(* IEC 61131-3 sources: HappyLearnCodesys/content/softmotion/CustomKinematics_Implementation, 3 files *)

(* ---- Jog.st ---- *)
(*
    檔案用途：
      封裝一個 Jog 功能塊，讓使用者可以同時在「軸空間（ACS）」與「笛卡兒空間（MCS）」下
      以按鍵方式點動 Gantry3C 自訂運動學的 TCP 位置。
    教學重點：
      - 利用兩個 SMC_GroupJog2 實例（jog_mcs、jog_axes）分別處理 TCP Jog 與關節 Jog。
      - 理解來自視覺介面的按鍵輸入（Jog_TCP_*、Jog_Drive_*）如何對應到 Forward/Backward 陣列。
      - 作為「自訂運動學上層 Jog 介面」的範例，可套用到其他 kinematics。
*)
/// This FB combines jogging in both axis space as well as cartesian space.
/// It uses two instances of SMC_GroupJog2. One for axis space and the other for cartesian space.
/// This FB can be used along with the visu templates V_RobotPosition_axes
/// and V_RobotPosition_cart_Jog to jog any kinematics in cartesian and axis space.

FUNCTION_BLOCK Jog
VAR_IN_OUT
	/// Reference to Axisgroup
	AxisGroup : AXIS_GROUP_REF_SM3;
END_VAR
VAR_INPUT
	/// Inputs (from the visu) to jog the robot in cartesian space
	Jog_TCP_Xp : BOOL;
	Jog_TCP_Xn : BOOL;
	Jog_TCP_Yp : BOOL;
	Jog_TCP_Yn : BOOL;
	Jog_TCP_Zp : BOOL;
	Jog_TCP_Zn : BOOL;
	Jog_TCP_Ap : BOOL;
	Jog_TCP_An : BOOL;
	Jog_TCP_Bp : BOOL;
	Jog_TCP_Bn : BOOL;
	Jog_TCP_Cp : BOOL;
	Jog_TCP_Cn : BOOL;

	/// Inputs (from the visu) to jog the robot in axis space
	Jog_Drive_Xp : BOOL;
	Jog_Drive_Xn : BOOL;
	Jog_Drive_Yp : BOOL;
	Jog_Drive_Yn : BOOL;
	Jog_Drive_Zp : BOOL;
	Jog_Drive_Zn : BOOL;
	Jog_Drive_Cp : BOOL;
	Jog_Drive_Cn : BOOL;

END_VAR
VAR
	/// SMC_GroupJog2 for cartesian space
	jog_mcs : SMC_GroupJog2 :=(Enable := TRUE, MaxLinearDistance := 2, MaxAngularDistance := 1,
							VelFactor := 1, AccFactor := 1, JerkFactor := 1,
							Velocity := 100, Acceleration := 1000, Deceleration := 1000, Jerk := 1000,
						    CoordSystem:= SMC_COORD_SYSTEM.MCS);

	/// SMC_GroupJog2 for axes space
	jog_axes : SMC_GroupJog2 :=(Enable := TRUE, MaxLinearDistance := 2, MaxAngularDistance := 1,
							VelFactor := 1, AccFactor := 1, JerkFactor := 1,
							Velocity := 100, Acceleration := 1000, Deceleration := 1000, Jerk := 1000,
						    CoordSystem:= SMC_COORD_SYSTEM.ACS);
END_VAR

jog_mcs.Forward[0] := Jog_TCP_Xp;
jog_mcs.Forward[1] := Jog_TCP_Yp;
jog_mcs.Forward[2] := Jog_TCP_Zp;
jog_mcs.Forward[3] := Jog_TCP_Ap;
jog_mcs.Forward[4] := Jog_TCP_Bp;
jog_mcs.Forward[5] := Jog_TCP_Cp;

jog_mcs.Backward[0] := Jog_TCP_Xn;
jog_mcs.Backward[1] := Jog_TCP_Yn;
jog_mcs.Backward[2] := Jog_TCP_Zn;
jog_mcs.Backward[3] := Jog_TCP_An;
jog_mcs.Backward[4] := Jog_TCP_Bn;
jog_mcs.Backward[5] := Jog_TCP_Cn;

jog_axes.Forward[0] := Jog_Drive_Xp;
jog_axes.Forward[1] := Jog_Drive_Yp;
jog_axes.Forward[2] := Jog_Drive_Zp;
jog_axes.Forward[3] := Jog_Drive_Cp;

jog_axes.Backward[0] := Jog_Drive_Xn;
jog_axes.Backward[1] := Jog_Drive_Yn;
jog_axes.Backward[2] := Jog_Drive_Zn;
jog_axes.Backward[3] := Jog_Drive_Cn;

jog_mcs(AxisGroup := Axisgroup);
jog_axes(AxisGroup := Axisgroup);

(* ---- SMC_TRAFOF_Gantry3C.st ---- *)
(*
    檔案用途：
      針對 Gantry3C 自訂運動學，將各軸的實際位置（DriveX/Y/Z/C）轉換為 TCP 位置（dx,dy,dz,dAzimuth），
      並依照設定的 min/max 範圍做正規化，方便在視覺模板中顯示。
    教學重點：
      - 理解 Offset（dOffset*）與 min/max 顯示範圍如何影響可視化座標。
      - 觀察正規化流程如何把實際座標壓縮到 -1..1 或類似比例，方便視窗呈現。
      - 作為自訂 Kinematics 用於視覺化轉換的範例，未牽涉運動控制本身。
*)
/// This FB transforms the input axes values of a Gantry3C Transformation to its respective TCP values.
/// Additionally the axes values are normalised to be used along with the visualization template
/// TRAFOF_Gantry3C_YZ to visualize the movements of the kinematics.
FUNCTION_BLOCK SMC_TRAFOF_Gantry3C
VAR_IN_OUT
    /// Reference to X-axis
    DriveX: AXIS_REF_SM3;
    /// Reference to Y-axis
    DriveY: AXIS_REF_SM3;
    /// Reference to Z-axis
    DriveZ: AXIS_REF_SM3;
    /// Reference to A-axis
    DriveC: AXIS_REF_SM3;
END_VAR
VAR_INPUT
    /// Offset position for X-axis
    dOffsetX:LREAL;
    /// Offset position for Y-axis
    dOffsetY:LREAL;
    /// Offset position for Z-axis
    dOffsetZ:LREAL;
    /// Offset position for A-axis
    dOffsetA:LREAL;
    /// Minimum display area of axis X for visualization
    minX:LREAL;
    /// Maximal display area of axis X for visualization
    maxX:LREAL;
    /// Minimum display area of axis Y for visualization
    minY:LREAL;
    /// Maximal display area of axis Y for visualization
    maxY:LREAL;
    /// Minimum display area of axis Z for visualization
	minZ:LREAL;
    /// Maximal display area of axis Z for visualization
	maxZ : LREAL;

END_VAR
VAR_OUTPUT
    /// position of the TCP in X axis
    dx: LREAL;
    /// position of the TCP in Y axis
    dy: LREAL;
    /// position of the TCP in Z axis
	dz: LREAL;
    /// position of the TCP in C axis
	dAzimuth:LREAL;
END_VAR
VAR
	/// normalised position
    dnx, dny, dnz:LREAL;
    dnxt, dnyt, dnzt:LREAL;
	sAz, cAz : LREAL;
    dm: LREAL;
END_VAR

dx:=DriveX.fActPosition-dOffsetX;
dy:=DriveY.fActPosition-dOffsetY;
dz:=DriveZ.fActPosition-dOffsetZ;
dAzimuth:=DriveC.fActPosition-dOffsetA;

sAz := SIN(dAzimuth/180.0*SMC_PI);
cAz := COS(dAzimuth/180.0*SMC_PI);

IF maxx > minx AND maxy > miny AND maxZ > minZ THEN
	dm := MAX(ABS(maxx), ABS(minx));
	dm := MAX(dm, ABS(maxy));
	dm := MAX(dm, ABS(miny));
	dm := MAX(dm, ABS(maxz));
	dm := MAX(dm, ABS(minz));

	dnx := (DriveX.fActPosition-dOffsetX)/dm;
	dny := (DriveY.fActPosition-dOffsetY)/dm;
	dnz := (DriveZ.fActPosition-dOffsetZ)/dm;

	dnxt := dx/dm;
	dnyt := dy/dm;
	dnzt := dz/dm;
END_IF

(* ---- Prg_Visu.st ---- *)
(*
    檔案用途：
      建立一個簡單的測試與視覺程式，用來驗證自訂 Gantry3C 運動學：
      - 啟動並啟用 AxisGroup；
      - 提供線性與直接移動指令（mla、mda）；
      - 呼叫 Jog FB 讓使用者在 MCS / ACS 中點動 TCP 或關節；
      - 呼叫 SMC_TRAFOF_Gantry3C 計算並正規化 TCP 位置，供視覺模板顯示。
    教學重點：
      - 將自訂 kinematics（Gantry3C）與 Jog、視覺化整合成一個可互動的測試環境。
      - 觀察 AxisGroup Power / Enable 流程與 jog、mla、mda 之間的關係。
*)
/// This is a simple program to test the Gantry3C kinematics.
/// The visualization can be used to Jog the robot(in axis and cartesian space) and command movements like
/// MC_MoveLinearAbsolute and MC_MoveDirectAbsolute.
/// The axisgroup will be powered and enabled immediately when the application is started so that the user
/// can start controlling the robot directly
PROGRAM Prg_Visu
VAR
	gpow : SMC_GroupPower :=(Enable := TRUE, bRegulatorOn := TRUE, bDriveStart := TRUE) ;
	gen : MC_GroupEnable;

	mla : MC_MoveLinearAbsolute :=(Velocity := 100, Acceleration := 1000, Deceleration := 1000, Jerk := 10000,
								   CoordSystem := SMC_COORD_SYSTEM.MCS);
	mda : MC_MoveDirectAbsolute :=(CoordSystem := SMC_COORD_SYSTEM.MCS);

	istate : INT;

	Gantry3C_Visu_Calc : SMC_TRAFOF_Gantry3C;
	jog : jog;

END_VAR

CASE istate OF
0:
	IF gpow.Status THEN
		gen.Execute := TRUE;
		istate := istate +10;
	END_IF
10:
	IF gen.Done THEN
		istate := istate +10;
	END_IF

END_CASE

gpow(AxisGroup := AxisGroup);
gen(AxisGroup := Axisgroup);
jog(AxisGroup := Axisgroup);
mla(AxisGroup := Axisgroup);
mda(Axisgroup := AxisGroup);
Gantry3C_Visu_Calc(	DriveX:= DriveX, DriveY:= DriveY, DriveZ:= DriveZ, DriveC:=DriveC,
					minX:= -10, maxX:= 500, minY:= -10, maxY:= 500, minZ := -10, maxZ := 500);
